// TIA Portal V18 export
// export: Created 2025-12-01T17:50:28.9556114Z, ExportSetting None, DisplayName Totally Integrated Automation Portal, DisplayVersion V18 Update 5, DisplayName TIA Portal Openness, DisplayVersion V18 Update 5, DisplayName TIA Portal Teamcenter Gateway, DisplayVersion V18, DisplayName TIA Portal Version Control Interface, DisplayVersion V18, DisplayName STEP 7 Professional, DisplayVersion V18 Update 5, DisplayName STEP 7 Safety, DisplayVersion V18, DisplayName WinCC Professional, DisplayVersion V18 Update 5
FUNCTION "CylinderModule_V2" : Void   // FC3010, LAD
TITLE = Title
{ S7_Optimized_Access := 'FALSE' }
VERSION : 2.0
// //---------------------------------------------------------------//
// //FunctionName:CylinderV2
// //FunctionDescription:CylinderControl
// //---------------------------------------------------------------//
// //in:
// 
// 	iReset	Bool			reset action
// 	iRun	Bool			system run
// 	iE_stop	Bool			e_stop monitor
// 	iManualMode	Bool		manual mode
// 	iAutoMode	Bool		auto mode
// 	iEnableAlarm	Bool		alarm will popup up
// 	iPulse_100mS	Bool		pulse *100ms
// 	iPulse_1S	Bool		pulse*1s
// 	iCyDBNO	Int	Int		Interface data block number
// 	iCyCounts	Int		total counts of cylinder to be used[must                                                                                                             be>=1 and <=100]
// 
// //inout:
// //out:
// //---------------------------------------------------------------//
// //Version:V2
// //D&T:2016-11-14
// //Group:RCS
// //Author:JM
// //-------------------------Modify1----------------------------------//
// //Version:
// //D&T:2016-11-17
// //Group: RCS
// //Author:
// //Modify:Update cylinder no as output interface
// //-------------------------Modify2----------------------------------//
// //Version:
// //D&T:2022-12-07
// //Group: RCS
// //Author:JM
// //Modify: add action time
// stored: AutoNumber false, SetENOAutomatically false
   VAR_INPUT
      iReset : Bool;   // reset action
      iRun : Bool;   // system run
      iEStop : Bool;   // e_stop monitor
      iManualMode : Bool;   // manual mode
      iAutoMode : Bool;   // auto mode
      iEnableAlarm : Bool;   // alarm will popup up
      iPulse100mS : Bool;   // pulse *100ms
      iPulse1S : Bool;   // pulse*1s
      iError : Bool;   // Outer error force output off
      iGoWorkInterlock : Bool;   // 1=permit motion
      iGoHomeInterlock : Bool;   // 1=permit motion
      iWorkPositionSensor : Bool;   // PLC DI
      iHomePositionSensor : Bool;   // PLC DI
      iValveType : Bool;   // reserve 2022-12-07 / 0 : don`t need holding(2way&3way middle sealing) / 1: need holding(3way middle leaking)
      iManualOutputType : Bool;   // 0 : Output not hold / 1: Output hold (in Manual mode)
      iFaultTime : Int;   // Value*100mS
      iOnPositionTime : Int;   // Value*100mS
   END_VAR
   VAR_OUTPUT
      oGoWP_ButtonActive : Bool;   // For HMI button,indicate can operate go work button
      oGoHP_ButtonActive : Bool;   // For HMI button,indicate can operate go home button
      oCyNo : Byte;
   END_VAR
   VAR_IN_OUT
      ioManualGoWork : Bool;
      ioManualGoHome : Bool;
      ioAutoGoWork : Bool;
      ioAutoGoHome : Bool;
      ioResetOut : Bool;
      ioGoWorkTime : Int;   // Time for going to work position
      ioGoHomeTime : Int;   // time for going to home position
      ioWorkFaultTime : Int;
      ioHomeFaultTime : Int;
      ioBothSensorOnTime : Int;
      ioPulse100mSP : Bool;
      ioAutoGoWorkP : Bool;
      ioAutoGoHomeP : Bool;
      ioGoWork100mSP : Bool;
      ioGoHome100mSP : Bool;
      ioBothSensorOn100mSP : Bool;
      ioAlarm : Bool;
      ioSpare1 : Bool;
      ioSpare2 : Byte;
      ioGoWorkFault : Bool;
      ioGoHomeFault : Bool;
      ioSensorPositionFault : Bool;
      ioGoWorkPosition : Bool;   // PLC DQ
      ioGoHomePosition : Bool;   // PLC DQ
   END_VAR
   VAR_TEMP   // added for the SCL form of the ladder/FBD networks
      _w1 : Bool;
      _w2 : Bool;
      _w3 : Bool;
      _w4 : Bool;
   END_VAR
BEGIN

REGION Network 1: Reset Go Work & Go Home
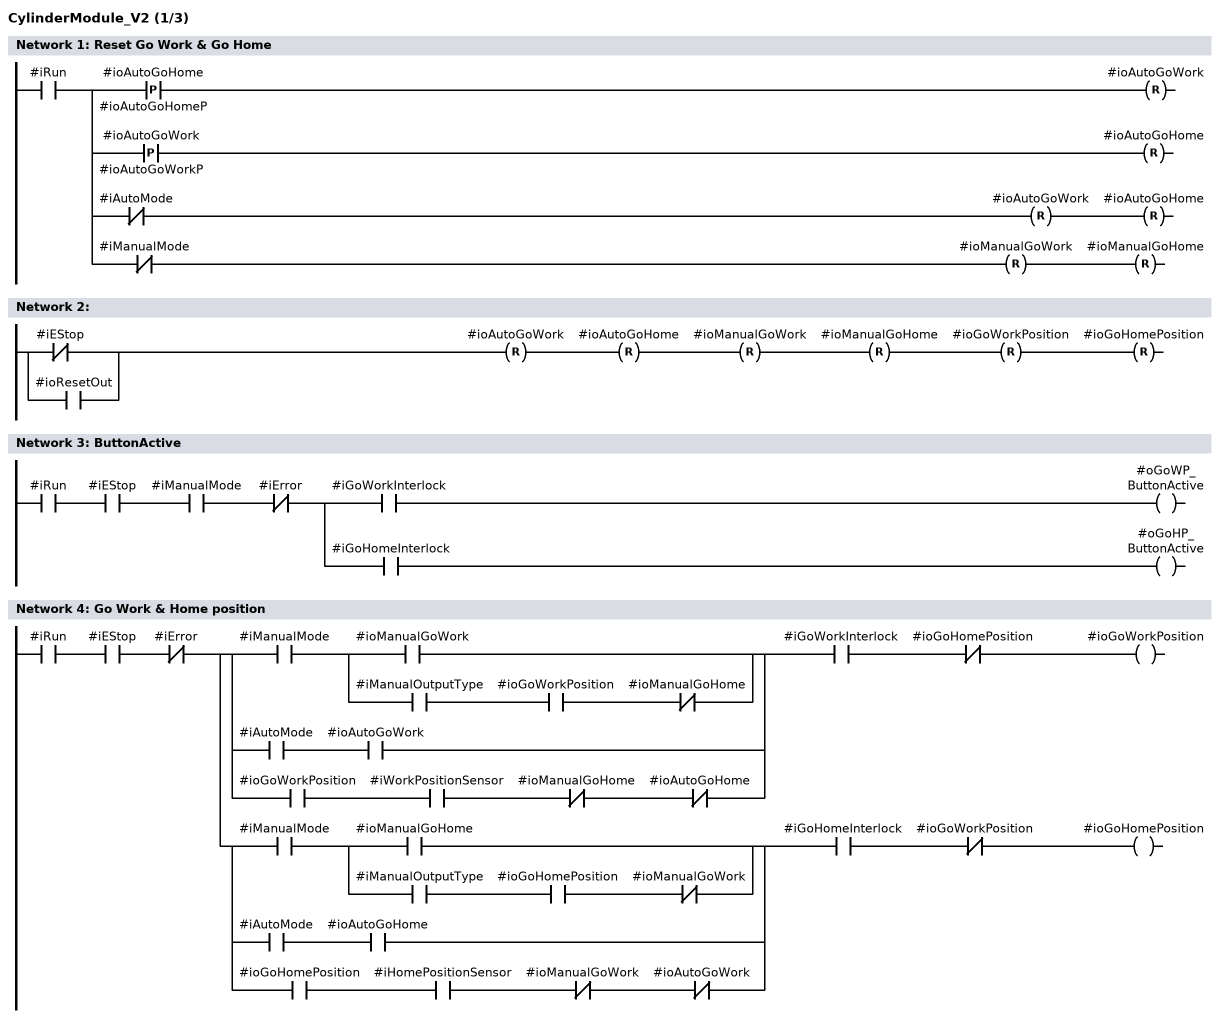
   RUNG wire#powerrail
      Contact( #iRun )
      wire#w1
      P_Contact(operand := #ioAutoGoHome, bit := #ioAutoGoHomeP)
      R_Coil( #ioAutoGoWork )
   END_RUNG
   RUNG wire#w1
      P_Contact(operand := #ioAutoGoWork, bit := #ioAutoGoWorkP)
      R_Coil( #ioAutoGoHome )
   END_RUNG
   RUNG wire#w1
      I_Contact( #iAutoMode )
      R_Coil( #ioAutoGoWork )
      R_Coil( #ioAutoGoHome )
   END_RUNG
   RUNG wire#w1
      I_Contact( #iManualMode )
      R_Coil( #ioManualGoWork )
      R_Coil( #ioManualGoHome )
   END_RUNG
   // the same network as SCL:
   #_w1 := #iRun AND #ioAutoGoHome AND NOT #ioAutoGoHomeP;   // rising edge of #ioAutoGoHome
   #ioAutoGoHomeP := #ioAutoGoHome;
   IF #_w1 THEN #ioAutoGoWork := FALSE; END_IF;
   #_w2 := #iRun AND #ioAutoGoWork AND NOT #ioAutoGoWorkP;   // rising edge of #ioAutoGoWork
   #ioAutoGoWorkP := #ioAutoGoWork;
   IF #_w2 THEN #ioAutoGoHome := FALSE; END_IF;
   IF #iRun AND NOT #iAutoMode THEN
       #ioAutoGoWork := FALSE;
       #ioAutoGoHome := FALSE;
   END_IF;
   IF #iRun AND NOT #iManualMode THEN
       #ioManualGoWork := FALSE;
       #ioManualGoHome := FALSE;
   END_IF;
END_REGION

REGION Network 2
   RUNG wire#powerrail
      I_Contact( #iEStop )
      wire#w1
      R_Coil( #ioAutoGoWork )
      R_Coil( #ioAutoGoHome )
      R_Coil( #ioManualGoWork )
      R_Coil( #ioManualGoHome )
      R_Coil( #ioGoWorkPosition )
      R_Coil( #ioGoHomePosition )
   END_RUNG
   RUNG wire#powerrail
      Contact( #ioResetOut )
   END_RUNG wire#w1
   // the same network as SCL:
   IF NOT #iEStop OR #ioResetOut THEN
       #ioAutoGoWork := FALSE;
       #ioAutoGoHome := FALSE;
       #ioManualGoWork := FALSE;
       #ioManualGoHome := FALSE;
       #ioGoWorkPosition := FALSE;
       #ioGoHomePosition := FALSE;
   END_IF;
END_REGION

REGION Network 3: ButtonActive
   RUNG wire#powerrail
      Contact( #iRun )
      Contact( #iEStop )
      Contact( #iManualMode )
      I_Contact( #iError )
      wire#w1
      Contact( #iGoWorkInterlock )
      Coil( #oGoWP_ButtonActive )
   END_RUNG
   RUNG wire#w1
      Contact( #iGoHomeInterlock )
      Coil( #oGoHP_ButtonActive )
   END_RUNG
   // the same network as SCL:
   #_w1 := #iRun AND #iEStop AND #iManualMode AND NOT #iError;
   #oGoWP_ButtonActive := #_w1 AND #iGoWorkInterlock;
   #oGoHP_ButtonActive := #_w1 AND #iGoHomeInterlock;
END_REGION

REGION Network 4: Go Work & Home position
   RUNG wire#powerrail
      Contact( #iRun )
      Contact( #iEStop )
      I_Contact( #iError )
      wire#w1
      Contact( #iManualMode )
      wire#w2
      Contact( #ioManualGoWork )
      wire#w3
      Contact( #iGoWorkInterlock )
      I_Contact( #ioGoHomePosition )
      Coil( #ioGoWorkPosition )
   END_RUNG
   RUNG wire#w2
      Contact( #iManualOutputType )
      Contact( #ioGoWorkPosition )
      I_Contact( #ioManualGoHome )
   END_RUNG wire#w3
   RUNG wire#w1
      Contact( #iAutoMode )
      Contact( #ioAutoGoWork )
   END_RUNG wire#w3
   RUNG wire#w1
      Contact( #ioGoWorkPosition )
      Contact( #iWorkPositionSensor )
      I_Contact( #ioManualGoHome )
      I_Contact( #ioAutoGoHome )
   END_RUNG wire#w3
   RUNG wire#w1
      Contact( #iManualMode )
      wire#w4
      Contact( #ioManualGoHome )
      wire#w5
      Contact( #iGoHomeInterlock )
      I_Contact( #ioGoWorkPosition )
      Coil( #ioGoHomePosition )
   END_RUNG
   RUNG wire#w4
      Contact( #iManualOutputType )
      Contact( #ioGoHomePosition )
      I_Contact( #ioManualGoWork )
   END_RUNG wire#w5
   RUNG wire#w1
      Contact( #iAutoMode )
      Contact( #ioAutoGoHome )
   END_RUNG wire#w5
   RUNG wire#w1
      Contact( #ioGoHomePosition )
      Contact( #iHomePositionSensor )
      I_Contact( #ioManualGoWork )
      I_Contact( #ioAutoGoWork )
   END_RUNG wire#w5
   // the same network as SCL:
   #_w1 := #iRun AND #iEStop AND NOT #iError;
   #ioGoWorkPosition := #_w1 AND ((#iManualMode AND (#ioManualGoWork OR (#iManualOutputType AND #ioGoWorkPosition AND NOT #ioManualGoHome))) OR (#iAutoMode AND #ioAutoGoWork) OR (#ioGoWorkPosition AND #iWorkPositionSensor AND NOT #ioManualGoHome AND NOT #ioAutoGoHome)) AND #iGoWorkInterlock AND NOT #ioGoHomePosition;
   #ioGoHomePosition := #_w1 AND ((#iManualMode AND (#ioManualGoHome OR (#iManualOutputType AND #ioGoHomePosition AND NOT #ioManualGoWork))) OR (#iAutoMode AND #ioAutoGoHome) OR (#ioGoHomePosition AND #iHomePositionSensor AND NOT #ioManualGoWork AND NOT #ioAutoGoWork)) AND #iGoHomeInterlock AND NOT #ioGoWorkPosition;
END_REGION

REGION Network 5: Go_work_fault
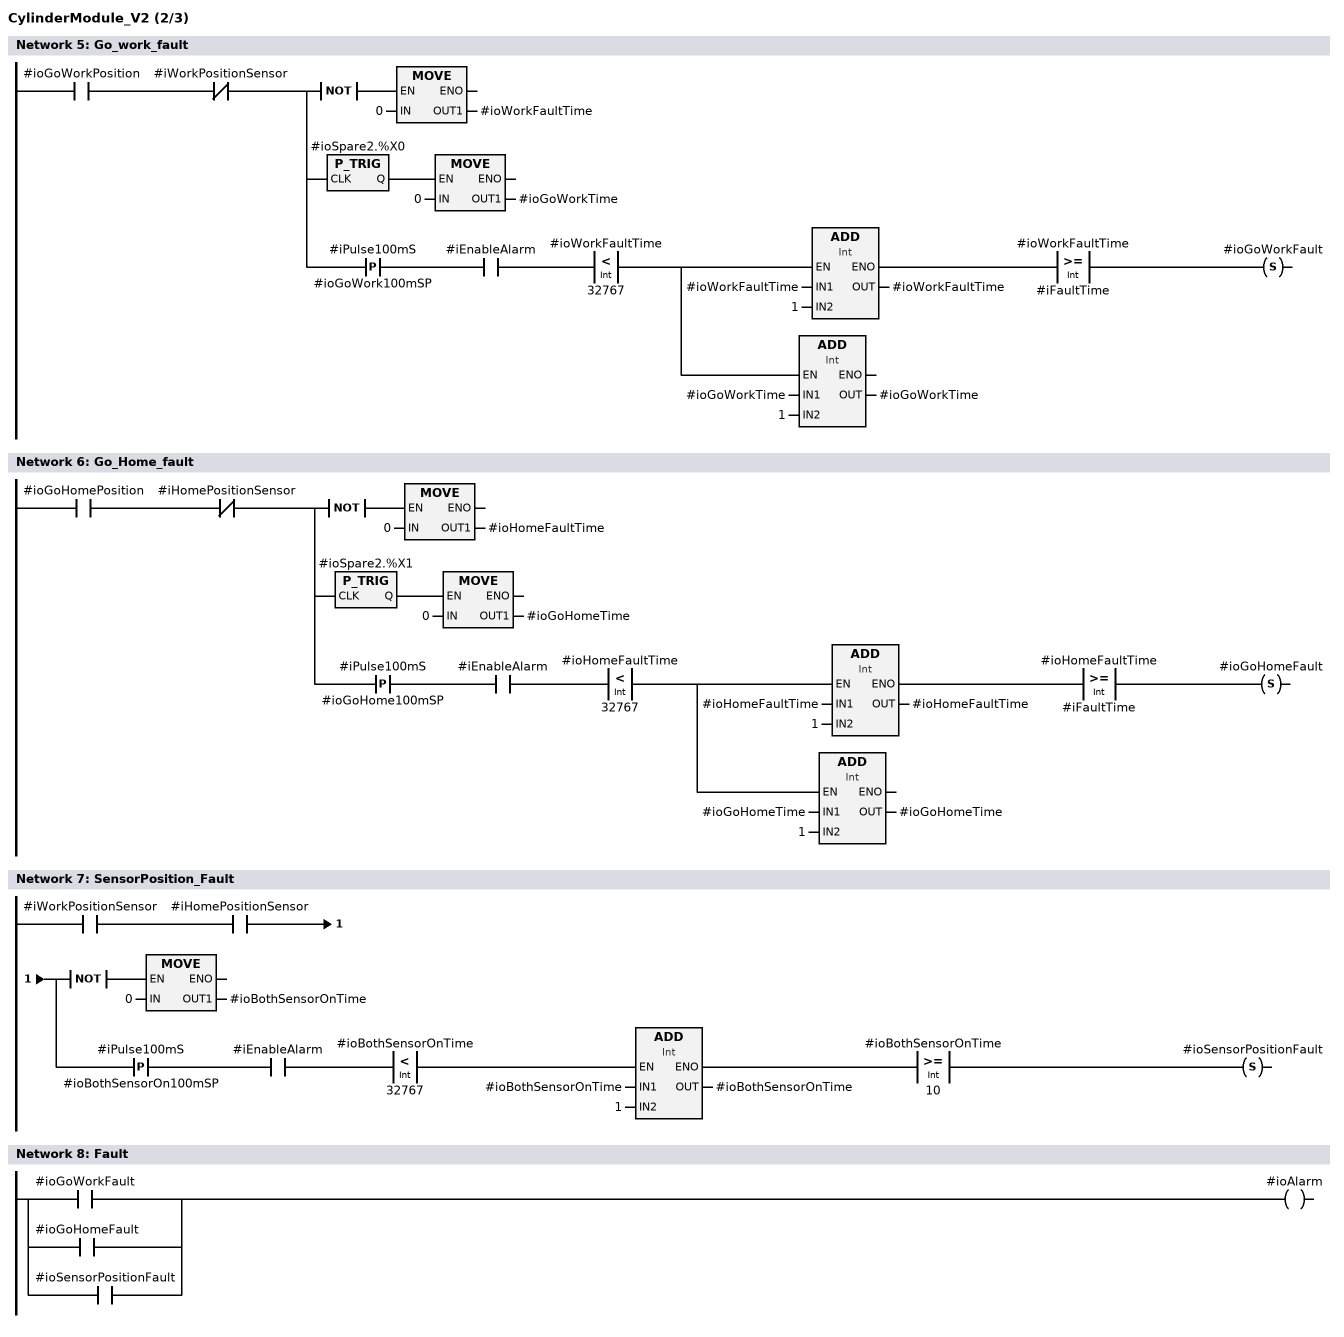
   RUNG wire#powerrail
      Contact( #ioGoWorkPosition )
      I_Contact( #iWorkPositionSensor )
      wire#w1
      Not()
      { S7_GenerateENO := "TRUE" } Move(in := 0, out1 => #ioWorkFaultTime)
   END_RUNG
   RUNG wire#w1
      P_Trig( #ioSpare2.%X0 )
      { S7_GenerateENO := "TRUE" } Move(in := 0, out1 => #ioGoWorkTime)
   END_RUNG
   RUNG wire#w1
      P_Contact(operand := #iPulse100mS, bit := #ioGoWork100mSP)
      Contact( #iEnableAlarm )
      { S7_Templates := "SrcType := Int" } LT_Contact(in1 := #ioWorkFaultTime, in2 := 32767)
      wire#w2
      { S7_Templates := "SrcType := Int"; S7_GenerateENO := "TRUE" } Add(in1 := #ioWorkFaultTime, in2 := 1, out => #ioWorkFaultTime)
      { S7_Templates := "SrcType := Int" } GE_Contact(in1 := #ioWorkFaultTime, in2 := #iFaultTime)
      S_Coil( #ioGoWorkFault )
   END_RUNG
   RUNG wire#w2
      { S7_Templates := "SrcType := Int"; S7_GenerateENO := "TRUE" } Add(in1 := #ioGoWorkTime, in2 := 1, out => #ioGoWorkTime)
   END_RUNG
   // the same network as SCL:
   // ENO of a box is taken as its EN; it also drops when the box reports an error
   #_w1 := #ioGoWorkPosition AND NOT #iWorkPositionSensor;
   IF NOT #_w1 THEN #ioWorkFaultTime := 0; END_IF;
   #_w2 := #_w1 AND NOT #ioSpare2.%X0;   // rising edge
   #ioSpare2.%X0 := #_w1;
   IF #_w2 THEN #ioGoWorkTime := 0; END_IF;
   #_w3 := #_w1 AND #iPulse100mS AND NOT #ioGoWork100mSP;   // rising edge of #iPulse100mS
   #ioGoWork100mSP := #iPulse100mS;
   #_w4 := #_w3 AND #iEnableAlarm AND (#ioWorkFaultTime < 32767);
   IF #_w4 THEN #ioWorkFaultTime := #ioWorkFaultTime + 1; END_IF;
   IF #_w4 AND (#ioWorkFaultTime >= #iFaultTime) THEN #ioGoWorkFault := TRUE; END_IF;
   IF #_w4 THEN #ioGoWorkTime := #ioGoWorkTime + 1; END_IF;
END_REGION

REGION Network 6: Go_Home_fault
   RUNG wire#powerrail
      Contact( #ioGoHomePosition )
      I_Contact( #iHomePositionSensor )
      wire#w1
      Not()
      { S7_GenerateENO := "TRUE" } Move(in := 0, out1 => #ioHomeFaultTime)
   END_RUNG
   RUNG wire#w1
      P_Trig( #ioSpare2.%X1 )
      { S7_GenerateENO := "TRUE" } Move(in := 0, out1 => #ioGoHomeTime)
   END_RUNG
   RUNG wire#w1
      P_Contact(operand := #iPulse100mS, bit := #ioGoHome100mSP)
      Contact( #iEnableAlarm )
      { S7_Templates := "SrcType := Int" } LT_Contact(in1 := #ioHomeFaultTime, in2 := 32767)
      wire#w2
      { S7_Templates := "SrcType := Int"; S7_GenerateENO := "TRUE" } Add(in1 := #ioHomeFaultTime, in2 := 1, out => #ioHomeFaultTime)
      { S7_Templates := "SrcType := Int" } GE_Contact(in1 := #ioHomeFaultTime, in2 := #iFaultTime)
      S_Coil( #ioGoHomeFault )
   END_RUNG
   RUNG wire#w2
      { S7_Templates := "SrcType := Int"; S7_GenerateENO := "TRUE" } Add(in1 := #ioGoHomeTime, in2 := 1, out => #ioGoHomeTime)
   END_RUNG
   // the same network as SCL:
   // ENO of a box is taken as its EN; it also drops when the box reports an error
   #_w1 := #ioGoHomePosition AND NOT #iHomePositionSensor;
   IF NOT #_w1 THEN #ioHomeFaultTime := 0; END_IF;
   #_w2 := #_w1 AND NOT #ioSpare2.%X1;   // rising edge
   #ioSpare2.%X1 := #_w1;
   IF #_w2 THEN #ioGoHomeTime := 0; END_IF;
   #_w3 := #_w1 AND #iPulse100mS AND NOT #ioGoHome100mSP;   // rising edge of #iPulse100mS
   #ioGoHome100mSP := #iPulse100mS;
   #_w4 := #_w3 AND #iEnableAlarm AND (#ioHomeFaultTime < 32767);
   IF #_w4 THEN #ioHomeFaultTime := #ioHomeFaultTime + 1; END_IF;
   IF #_w4 AND (#ioHomeFaultTime >= #iFaultTime) THEN #ioGoHomeFault := TRUE; END_IF;
   IF #_w4 THEN #ioGoHomeTime := #ioGoHomeTime + 1; END_IF;
END_REGION

REGION Network 7: SensorPosition_Fault
   RUNG wire#powerrail
      Contact( #iWorkPositionSensor )
      Contact( #iHomePositionSensor )
      wire#w1
      Not()
      { S7_GenerateENO := "TRUE" } Move(in := 0, out1 => #ioBothSensorOnTime)
   END_RUNG
   RUNG wire#w1
      P_Contact(operand := #iPulse100mS, bit := #ioBothSensorOn100mSP)
      Contact( #iEnableAlarm )
      { S7_Templates := "SrcType := Int" } LT_Contact(in1 := #ioBothSensorOnTime, in2 := 32767)
      { S7_Templates := "SrcType := Int"; S7_GenerateENO := "TRUE" } Add(in1 := #ioBothSensorOnTime, in2 := 1, out => #ioBothSensorOnTime)
      { S7_Templates := "SrcType := Int" } GE_Contact(in1 := #ioBothSensorOnTime, in2 := 10)
      S_Coil( #ioSensorPositionFault )
   END_RUNG
   // the same network as SCL:
   // ENO of a box is taken as its EN; it also drops when the box reports an error
   #_w1 := #iWorkPositionSensor AND #iHomePositionSensor;
   IF NOT #_w1 THEN #ioBothSensorOnTime := 0; END_IF;
   #_w2 := #_w1 AND #iPulse100mS AND NOT #ioBothSensorOn100mSP;   // rising edge of #iPulse100mS
   #ioBothSensorOn100mSP := #iPulse100mS;
   #_w3 := #_w2 AND #iEnableAlarm AND (#ioBothSensorOnTime < 32767);
   IF #_w3 THEN #ioBothSensorOnTime := #ioBothSensorOnTime + 1; END_IF;
   IF #_w3 AND (#ioBothSensorOnTime >= 10) THEN #ioSensorPositionFault := TRUE; END_IF;
END_REGION

REGION Network 8: Fault
   RUNG wire#powerrail
      Contact( #ioGoWorkFault )
      wire#w1
      Coil( #ioAlarm )
   END_RUNG
   RUNG wire#powerrail
      Contact( #ioGoHomeFault )
   END_RUNG wire#w1
   RUNG wire#powerrail
      Contact( #ioSensorPositionFault )
   END_RUNG wire#w1
   // the same network as SCL:
   #ioAlarm := #ioGoWorkFault OR #ioGoHomeFault OR #ioSensorPositionFault;
END_REGION

REGION Network 9: Reset fault
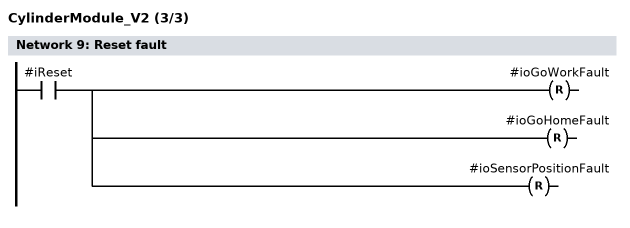
   RUNG wire#powerrail
      Contact( #iReset )
      wire#w1
      R_Coil( #ioGoWorkFault )
   END_RUNG
   RUNG wire#w1
      R_Coil( #ioGoHomeFault )
   END_RUNG
   RUNG wire#w1
      R_Coil( #ioSensorPositionFault )
   END_RUNG
   // the same network as SCL:
   IF #iReset THEN
       #ioGoWorkFault := FALSE;
       #ioGoHomeFault := FALSE;
       #ioSensorPositionFault := FALSE;
   END_IF;
END_REGION
END_FUNCTION
